Staubli VAL3: jointToArray.pgx

public program jointToArray(jointRx& x_jJointInput[], num& x_nNumOutput[])
  local jointRx l_jJointInput
begin

  //==========解析两个机器人之间通讯收发的数据和指令==========

  //将机器人的关节位置解析成数组格式
  l_jJointInput=x_jJointInput

  x_nNumOutput[0]=l_jJointInput.j1
  x_nNumOutput[1]=l_jJointInput.j2
  x_nNumOutput[2]=l_jJointInput.j3
  x_nNumOutput[3]=l_jJointInput.j4
  x_nNumOutput[4]=l_jJointInput.j5
  x_nNumOutput[5]=l_jJointInput.j6

  //将机器人的笛卡尔位置解析成数组格式

end
